# EPICS autosave request: iocBoot/ioc13bmc_linux/XPS_positions.req
file "CARS_8_motor_positions_sub.req",  P=$(P), M1=m33, M2=m34, M3=m35, M4=m36, M5=m37, M6=m38, M7=m39, M8=m40
file "CARS_motor_positions.req",        P=$(P), M=m41
file "CARS_motor_positions.req",        P=$(P), M=m42
file "CARS_motor_positions.req",        P=$(P), M=m43
file "CARS_motor_positions.req",        P=$(P), M=m44
file "CARS_motor_positions.req",        P=$(P), M=m45
file "CARS_motor_positions.req",        P=$(P), M=m46
